# EPICS StreamDevice protocol: epics/magnets.proto
# ./dtwinApp/Db/magnets.proto
Terminator = CR LF;

get_MBH2I00H { out "MBH2I00H.BDL?"; in "MBH2I00H.BDL %f"; ExtraInput = Ignore; }
set_MBH2I00H { out "MBH2I00H.BDL %f"; ExtraInput = Ignore; @init { get_MBH2I00H; } }

get_MBH2I00V { out "MBH2I00V.BDL?"; in "MBH2I00V.BDL %f"; ExtraInput = Ignore; }
set_MBH2I00V { out "MBH2I00V.BDL %f"; ExtraInput = Ignore; @init { get_MBH2I00V; } }

get_MBH2I00AH { out "MBH2I00AH.BDL?"; in "MBH2I00AH.BDL %f"; ExtraInput = Ignore; }
set_MBH2I00AH { out "MBH2I00AH.BDL %f"; ExtraInput = Ignore; @init { get_MBH2I00AH; } }

get_MBH2I00AV { out "MBH2I00AV.BDL?"; in "MBH2I00AV.BDL %f"; ExtraInput = Ignore; }
set_MBH2I00AV { out "MBH2I00AV.BDL %f"; ExtraInput = Ignore; @init { get_MBH2I00AV; } }

get_MFX2I01_US { out "MFX2I01_US.BDL?"; in "MFX2I01_US.BDL %f"; ExtraInput = Ignore; }
set_MFX2I01_US { out "MFX2I01_US.BDL %f"; ExtraInput = Ignore; @init { get_MFX2I01_US; } }

get_MFX2I01_DS { out "MFX2I01_DS.BDL?"; in "MFX2I01_DS.BDL %f"; ExtraInput = Ignore; }
set_MFX2I01_DS { out "MFX2I01_DS.BDL %f"; ExtraInput = Ignore; @init { get_MFX2I01_DS; } }

get_MBH2I01H { out "MBH2I01H.BDL?"; in "MBH2I01H.BDL %f"; ExtraInput = Ignore; }
set_MBH2I01H { out "MBH2I01H.BDL %f"; ExtraInput = Ignore; @init { get_MBH2I01H; } }

get_MBH2I01V { out "MBH2I01V.BDL?"; in "MBH2I01V.BDL %f"; ExtraInput = Ignore; }
set_MBH2I01V { out "MBH2I01V.BDL %f"; ExtraInput = Ignore; @init { get_MBH2I01V; } }

get_MBH2I01AH { out "MBH2I01AH.BDL?"; in "MBH2I01AH.BDL %f"; ExtraInput = Ignore; }
set_MBH2I01AH { out "MBH2I01AH.BDL %f"; ExtraInput = Ignore; @init { get_MBH2I01AH; } }

get_MBH2I01AV { out "MBH2I01AV.BDL?"; in "MBH2I01AV.BDL %f"; ExtraInput = Ignore; }
set_MBH2I01AV { out "MBH2I01AV.BDL %f"; ExtraInput = Ignore; @init { get_MBH2I01AV; } }

get_MBH1I02H { out "MBH1I02H.BDL?"; in "MBH1I02H.BDL %f"; ExtraInput = Ignore; }
set_MBH1I02H { out "MBH1I02H.BDL %f"; ExtraInput = Ignore; @init { get_MBH1I02H; } }

get_MBH1I02V { out "MBH1I02V.BDL?"; in "MBH1I02V.BDL %f"; ExtraInput = Ignore; }
set_MBH1I02V { out "MBH1I02V.BDL %f"; ExtraInput = Ignore; @init { get_MBH1I02V; } }

get_MFX1I03_US { out "MFX1I03_US.BDL?"; in "MFX1I03_US.BDL %f"; ExtraInput = Ignore; }
set_MFX1I03_US { out "MFX1I03_US.BDL %f"; ExtraInput = Ignore; @init { get_MFX1I03_US; } }

get_MFX1I03_DS { out "MFX1I03_DS.BDL?"; in "MFX1I03_DS.BDL %f"; ExtraInput = Ignore; }
set_MFX1I03_DS { out "MFX1I03_DS.BDL %f"; ExtraInput = Ignore; @init { get_MFX1I03_DS; } }

get_MBH1I03H { out "MBH1I03H.BDL?"; in "MBH1I03H.BDL %f"; ExtraInput = Ignore; }
set_MBH1I03H { out "MBH1I03H.BDL %f"; ExtraInput = Ignore; @init { get_MBH1I03H; } }

get_MBH1I03V { out "MBH1I03V.BDL?"; in "MBH1I03V.BDL %f"; ExtraInput = Ignore; }
set_MBH1I03V { out "MBH1I03V.BDL %f"; ExtraInput = Ignore; @init { get_MBH1I03V; } }

get_MQW1I03 { out "MQW1I03.BDL?"; in "MQW1I03.BDL %f"; ExtraInput = Ignore; }
set_MQW1I03 { out "MQW1I03.BDL %f"; ExtraInput = Ignore; @init { get_MQW1I03; } }

get_MQW1I04 { out "MQW1I04.BDL?"; in "MQW1I04.BDL %f"; ExtraInput = Ignore; }
set_MQW1I04 { out "MQW1I04.BDL %f"; ExtraInput = Ignore; @init { get_MQW1I04; } }

get_MBH1I04H { out "MBH1I04H.BDL?"; in "MBH1I04H.BDL %f"; ExtraInput = Ignore; }
set_MBH1I04H { out "MBH1I04H.BDL %f"; ExtraInput = Ignore; @init { get_MBH1I04H; } }

get_MBH1I04V { out "MBH1I04V.BDL?"; in "MBH1I04V.BDL %f"; ExtraInput = Ignore; }
set_MBH1I04V { out "MBH1I04V.BDL %f"; ExtraInput = Ignore; @init { get_MBH1I04V; } }

get_MFG1I04A { out "MFG1I04A.BDL?"; in "MFG1I04A.BDL %f"; ExtraInput = Ignore; }
set_MFG1I04A { out "MFG1I04A.BDL %f"; ExtraInput = Ignore; @init { get_MFG1I04A; } }

get_MFG1I04B { out "MFG1I04B.BDL?"; in "MFG1I04B.BDL %f"; ExtraInput = Ignore; }
set_MFG1I04B { out "MFG1I04B.BDL %f"; ExtraInput = Ignore; @init { get_MFG1I04B; } }

get_MBH1I05H { out "MBH1I05H.BDL?"; in "MBH1I05H.BDL %f"; ExtraInput = Ignore; }
set_MBH1I05H { out "MBH1I05H.BDL %f"; ExtraInput = Ignore; @init { get_MBH1I05H; } }

get_MBH1I05V { out "MBH1I05V.BDL?"; in "MBH1I05V.BDL %f"; ExtraInput = Ignore; }
set_MBH1I05V { out "MBH1I05V.BDL %f"; ExtraInput = Ignore; @init { get_MBH1I05V; } }

get_MQW1I05 { out "MQW1I05.BDL?"; in "MQW1I05.BDL %f"; ExtraInput = Ignore; }
set_MQW1I05 { out "MQW1I05.BDL %f"; ExtraInput = Ignore; @init { get_MQW1I05; } }

get_MQW1I06 { out "MQW1I06.BDL?"; in "MQW1I06.BDL %f"; ExtraInput = Ignore; }
set_MQW1I06 { out "MQW1I06.BDL %f"; ExtraInput = Ignore; @init { get_MQW1I06; } }

get_MBH1I07H { out "MBH1I07H.BDL?"; in "MBH1I07H.BDL %f"; ExtraInput = Ignore; }
set_MBH1I07H { out "MBH1I07H.BDL %f"; ExtraInput = Ignore; @init { get_MBH1I07H; } }

get_MBH1I07V { out "MBH1I07V.BDL?"; in "MBH1I07V.BDL %f"; ExtraInput = Ignore; }
set_MBH1I07V { out "MBH1I07V.BDL %f"; ExtraInput = Ignore; @init { get_MBH1I07V; } }

get_MFX0I01_US { out "MFX0I01_US.BDL?"; in "MFX0I01_US.BDL %f"; ExtraInput = Ignore; }
set_MFX0I01_US { out "MFX0I01_US.BDL %f"; ExtraInput = Ignore; @init { get_MFX0I01_US; } }

get_MFX0I01_DS { out "MFX0I01_DS.BDL?"; in "MFX0I01_DS.BDL %f"; ExtraInput = Ignore; }
set_MFX0I01_DS { out "MFX0I01_DS.BDL %f"; ExtraInput = Ignore; @init { get_MFX0I01_DS; } }

get_MBH0I01H { out "MBH0I01H.BDL?"; in "MBH0I01H.BDL %f"; ExtraInput = Ignore; }
set_MBH0I01H { out "MBH0I01H.BDL %f"; ExtraInput = Ignore; @init { get_MBH0I01H; } }

get_MBH0I01V { out "MBH0I01V.BDL?"; in "MBH0I01V.BDL %f"; ExtraInput = Ignore; }
set_MBH0I01V { out "MBH0I01V.BDL %f"; ExtraInput = Ignore; @init { get_MBH0I01V; } }

get_MHD0I01AH { out "MHD0I01AH.BDL?"; in "MHD0I01AH.BDL %f"; ExtraInput = Ignore; }
set_MHD0I01AH { out "MHD0I01AH.BDL %f"; ExtraInput = Ignore; @init { get_MHD0I01AH; } }

get_MHD0I01AV { out "MHD0I01AV.BDL?"; in "MHD0I01AV.BDL %f"; ExtraInput = Ignore; }
set_MHD0I01AV { out "MHD0I01AV.BDL %f"; ExtraInput = Ignore; @init { get_MHD0I01AV; } }

get_MBH0I01BH { out "MBH0I01BH.BDL?"; in "MBH0I01BH.BDL %f"; ExtraInput = Ignore; }
set_MBH0I01BH { out "MBH0I01BH.BDL %f"; ExtraInput = Ignore; @init { get_MBH0I01BH; } }

get_MBH0I01BV { out "MBH0I01BV.BDL?"; in "MBH0I01BV.BDL %f"; ExtraInput = Ignore; }
set_MBH0I01BV { out "MBH0I01BV.BDL %f"; ExtraInput = Ignore; @init { get_MBH0I01BV; } }
